Staubli VAL3: WAIT.pjx

--- WAIT.pjx ---
Parameters version=s7.5 stackSize=5000 millimeterUnit=true
Program file=condition.pgx
Program file=find.pgx
Program file=get.pgx
Program file=getSize.pgx
Program file=getType.pgx
Program file=isActive.pgx
Program file=load.pgx
Program file=make_it.pgx
Program file=onEdit.pgx
Program file=onInsert.pgx
Program file=onProgEnd.pgx
Program file=onRun.pgx
Program file=onStart.pgx
Program file=onStop.pgx
Program file=selectType.pgx
Program file=stopRobot.pgx
Data file=WAIT.dtx
Library alias=use path=Disk://kernel/userPage/userPage.pjx
Library alias=cycleStatus path=Disk://cycleStatus/cycleStatus.pjx
Library alias=language path=Disk://kernel/language/language.pjx
Library alias=saveInOut path=Disk://saveInputOutput/saveInputOutput.pjx
Type name=aioItem path=Disk://kernel/template/aioItem/aioItem.pjx
Type name=countItem path=Disk://kernel/template/countItem/countItem.pjx

--- find.pgx ---
public program find(string& x_sItem[], bool& x_bFound[])
  local num l_nIndex
  local num l_nOperator
  local num l_nValue
  local string l_sItem[2]
begin
  // REMOVE THE COUNT
  x_sItem=right(x_sItem,len(x_sItem)-len("WAIT "))
  // look inside
  x_bFound=isDefined(saveInOut:cCount[x_sItem])
  if !x_bFound
    x_bFound=isDefined(saveInOut:aCount[x_sItem])
  endIf
end

--- get.pgx ---
public program get(string& x_sItem[], num x_nIndex)
  local string l_sKey
  local num i
begin
  // OUTPUT
  // start from the first
  l_sKey=first(saveInOut:cCount)
  // search it
  while l_sKey!=""
    x_sItem=l_sKey
    l_sKey=next(saveInOut:cCount[l_sKey])
    if i==x_nIndex
      return
    else
      i=i+1
    endIf
  endWhile
  // start from the first
  l_sKey=first(saveInOut:aCount)
  while l_sKey!=""
    x_sItem=l_sKey
    l_sKey=next(saveInOut:aCount[l_sKey])
    if i==x_nIndex
      return
    else
      i=i+1
    endIf
  endWhile
end

--- getSize.pgx ---
public program getSize(num& x_nSize[])
begin
  // get the size for the counter
  x_nSize=size(saveInOut:cCount)
  // get the size for the aCounter
  x_nSize=x_nSize+size(saveInOut:aCount)
end

--- make_it.pgx ---
program make_it(string& x_sItem)
  local string l_sMessage
  local num i
  local num l_nValue
  local string l_sEmpty
  local string l_sItem
  local num l_nSizeList
  local string l_sEvent
  local bool l_bActive
  local string l_sItemList
  local num l_nKey
  local num l_nIndex
  local string l_sButton[2]
  local bool l_bYes
begin
  //
  cls()
  // Select the operator
  call language:message(l_sMessage,110)
  call use:questionDialog(l_sMessage,saveInOut:sCondition,i)
  //
  // != >= > < <= ==
  // compose the istruction
  if i>=1 and i<=size(saveInOut:sCondition)
    x_sItem=x_sItem+saveInOut:sCondition[i-1]
  else
    // escape
    x_sItem=""
    return
  endIf
  // modify the actual item
  call use:type(2,12,x_sItem)
  // insert a value
  call language:message(l_sMessage,112)
  // get the yes_no button Key
  call language:getYesNo(l_sButton)
  // ask the question
  call use:yes_no(l_sMessage,l_sButton,l_bYes)
  // check it
  if l_bYes
    //
    // reuse the operator
    //
    call saveInOut:getSize_num(l_nSizeList)
    call getType(l_sItem)
    call use:setSizeList(21,0,17,10)
    call use:listcreate(l_sItem)
    // insert in the list
    for i=0 to l_nSizeList-1
      call saveInOut:get_num(l_sItemList,i)
      call isActive(l_bActive,l_sItemList)
      if l_bActive
        call use:listadd(l_sItemList)
      endIf
    endFor
    call use:listredraw(0)
    do
      // get the key
      l_nKey=get()
      // get one input from the list
      call use:listevent(l_nKey,l_nIndex,l_sEvent)
      if l_nKey==255
        return
      endIf
    until l_nKey==270
    // check if an item has been selected
    if l_sEvent==""
      x_sItem=""
      return
    else
      x_sItem=x_sItem+l_sEvent
    endIf
  else
    // use a value
    call use:changeValue(l_nValue,-10000,10000,2+len(x_sItem),12,l_sEmpty)
    x_sItem=x_sItem+toString("",l_nValue)
  endIf
  // validate
  if use:bUseEscape
    x_sItem=""
  endIf
end

--- onEdit.pgx ---
public program onEdit(string& x_sItem[])
  local num l_nX
  local num l_nY
  local num l_nDelay
  local bool l_bValide
  local num l_nIndex
  local num l_nOperator
  local num l_nValue
  local string l_sType
  local string l_sName
begin
  // decompose it
  call saveInOut:decompose_wait(x_sItem,l_sName,l_nOperator,l_nValue)
  if l_sName!=""
    // get the item
    call saveInOut:get_num(x_sItem,l_nIndex)
    // edit it
    call make_it(x_sItem)
  else
    x_sItem=""
  endIf
end

--- onInsert.pgx ---
public program onInsert(string& x_sItem[])
  local string l_sEvent
begin
  cls()
  // select the type
  call selectType(l_sEvent)
  // exit
  if l_sEvent==""
    return
  else
    // copy it
    x_sItem=l_sEvent
  endIf
  // make it
  call make_it(x_sItem)
  //
end

--- onRun.pgx ---
public program onRun(string& x_sItem[])
  local num l_nValue
  local bool l_bCheck
  local num l_nIndex
  local num l_nOperator
  local string l_sName
begin
  // decompose
  call saveInOut:decompose_wait(x_sItem,l_sName,l_nOperator,l_nValue)
  if l_nIndex!=-1
    // check
    call condition(l_nOperator,l_nValue,l_sName,l_bCheck)
    // stop the robot
    if !l_bCheck
      call stopRobot()
      // <> >= > < <= ==
      do
        call condition(l_nOperator,l_nValue,l_sName,l_bCheck)
        delay(0)
      until l_bCheck==true
      // restart the robot
      cycleStatus:bWait=false
    endIf
  endIf
end

--- selectType.pgx ---
program selectType(string& x_sItem)
  local num l_nSizeList
  local string l_sItem
  local bool l_bActive
  local string l_sItemList
  local string l_sMessage
  local num l_nKey
  local string l_sEvent
  local num l_nSize
  local num i
  local string l_sName
begin
  // CNT
  call saveInOut:getSize_num(l_nSizeList)
  call getType(l_sItem)
  l_nSize=0
  //
  // create the list
  //
  call use:setSizeList(19,0,19,11)
  call use:listcreate(l_sItem)
  // insert in the list
  for i=0 to l_nSizeList-1
    call saveInOut:get_num(l_sItemList,i)
    call isActive(l_bActive,l_sItemList)
    if l_bActive
      call saveInOut:get_num(l_sItemList,i)
      call saveInOut:getItem_num(l_sName,l_sItemList)
      l_sItemList=l_sItemList+" {"+l_sName+"}"
      call use:listadd(l_sItemList)
    endIf
  endFor
  call use:selectNewField(nIndex,nIndex,0)
  call use:clear(0,13)
  call language:message(l_sMessage,63)
  call use:typeCenter(13,l_sMessage,40,true)
  do
    // get the key
    l_nKey=get()
    // get one input from the list
    call use:listevent(l_nKey,nIndex,l_sEvent)
    if l_nKey==255
      return
    endIf
  until l_nKey==270
  // save it
  if l_sEvent!=""
    x_sItem=left(l_sEvent,find(l_sEvent,"{")-1)
  else
    x_sItem=""
  endIf
end
